// TIA Portal V18 export
TYPE "hmi_home_1"
// stored: IsFailsafeCompliant false
   STRUCT
      pos : Real;
      eF : Bool;
      eR : Bool;
      mF : Bool;
      mR : Bool;
   END_STRUCT;
END_TYPE
